FUNCTION_BLOCK TcoLoggerSinkConfiguration 

VAR_INPUT
	Config		: REFERENCE TO TcoLoggerConfiguration;
END_VAR

VAR
	_xaeSink		: AdsLogSink;
	_volatileSink	: VolatileSink;
END_VAR

METHOD PUBLIC Memory : REFERENCE TO TcoLoggerConfiguration
VAR_INPUT
END_VAR
Config.AddSink(_volatileSink);
Memory REF= Config;
END_METHOD

METHOD PUBLIC XAE : REFERENCE TO TcoLoggerConfiguration
VAR_INPUT
END_VAR
Config.AddSink(_xaeSink);
XAE := Config;
END_METHOD

END_FUNCTION_BLOCK

(* stored: Version 1.1.0.1, ProductVersion 3.1.4024.9
   POU TcoLoggerSinkConfiguration: Id {e272c544-e71c-03a0-0b60-a798d7eaaffa}, SpecialFunc None
   Method Memory: Id {50b0a892-7347-0f8e-1e32-74a8a731b1a5}
   Method XAE: Id {66c0f21a-b76d-0a03-1dcf-41f50e56eb96} *)
